FUNCTION_BLOCK fb_CSVRead
VAR_INPUT
	bExecute:BOOL;
	dbid:UINT;
	table:STRING(100);
END_VAR
VAR_OUTPUT
	bError:BOOL:=FALSE;
	bReady:BOOL:=FALSE;
END_VAR
VAR
	PLCDBRead:fb_PLCDBRead(sNetid:='', tTimeOut:=T#15S);
	ReadStruct: ARRAY [0..1700] OF ST_ReturnedData;
	Columnnames: ARRAY [0..4] OF STRING(50):=['Dátum', 'temp_set', 'temp_act', 'hum_set', 'hum_act'];
END_VAR

IF bExecute THEN
	IF PLCDBread.ReadStruct(hDBID:=dbid,
							sTableName:=table,
							pColumnNames:=ADR(ColumnNames),
							cbColumnNames:=SIZEOF(ColumnNames),
							sOrderByColumn:='Dátum',
							eOrderType:=E_ordertype.ASC,
							nStartIndex:=0,
							nRecordCount:=1000,
							pData:=ADR(readstruct),
							cbData:=SIZEOF(readstruct))
	THEN
	IF plcdbread.bError THEN
		berror:=TRUE;	
	ELSE
	IF NOT plcdbread.bBusy THEN
		bExecute:=FALSE;
		bReady:=TRUE;
	END_IF	
	END_IF
	END_IF				
END_IF

METHOD ClearArray : BOOL
VAR_INPUT
END_VAR
memset(adr(readstruct),0,sizeof(readstruct));
END_METHOD

METHOD reset : BOOL
VAR_INPUT
END_VAR
bReady:=false;
END_METHOD

END_FUNCTION_BLOCK

(* stored: Version 1.1.0.1, ProductVersion 3.1.4024.2
   POU fb_CSVRead: Id {659727eb-0be6-4836-bb55-8234476a08aa}, SpecialFunc None
   Method ClearArray: Id {585624b8-a82f-4907-9741-f081bc9d50e4}
   Method reset: Id {0f71b593-3e49-43a6-966a-d876fcd12cb8} *)
